{attribute addProperty BoxType "AX8118-0000-0100-0100"}
{attribute addProperty Id "DeviceDevice_F82A60211620Ch_ACh_A_359CD49A176220WcStateAT %I*WcState_98A4DF7520.250InfoDataAT %I*InfoData_F030DC9B200250"}
{attribute addProperty CRC "2011418308"}
{attribute addProperty SizeInBites "394"}
{attribute addProperty SizeInBytes "49.25"}
TYPE AX8118_6822C7B9 :
STRUCT
	{attribute addProperty Name "Device"}
	Device : Device_F82A6021;
	{attribute addProperty Name "Ch_A"}
	Ch_A : Ch_A_359CD49A;
	{attribute addProperty Name "WcState"}
	WcState : WcState_98A4DF75;
	{attribute addProperty Name "InfoData"}
	InfoData : InfoData_F030DC9B;
END_STRUCT
END_TYPE

(* stored: Version 1.2.0.0, ProductVersion 3.1.4024.9
   DUT AX8118_6822C7B9: Id {b6a64542-2065-4d9a-bdf8-ed0d79b14b27} *)
